PROGRAM MAIN
VAR
END_VAR

FC_Instances();

END_PROGRAM

(* stored: Version 1.1.0.1
   POU MAIN: Id {c524df1f-557d-4d27-961d-2b5d2a6397cf}, SpecialFunc None *)
